FUNCTION_BLOCK AX_RF_TRIG (* Boolean falling and rising edge detection *)
  (* Standard: 61499-1 Annex A; Description: Copyright (c) 2017 fortiss GmbH, HR Agrartechnik GmbH This program and the accompanying materials are made available under the terms of the Eclipse Public License 2.0 which is available at https://www.eclipse.org/legal/epl-2.0/ SPDX-License-Identifier: EPL-2.0 *)
  (* Version 1.0, 2026-05-08, Franz Höpfinger, HR Agrartechnik GmbH, initial API and implementation and/or initial documentation *)
  PACKAGE adapter::events::unidirectional;
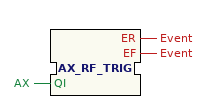
  EVENT_OUTPUT
    ER; (* confirmation that a rising edge was detected *)
    EF; (* confirmation that a falling edge was detected *)
  END_EVENT
  SOCKETS
    QI : adapter::types::unidirectional::AX; (* value to check for a rising or falling edge *)
  END_SOCKETS
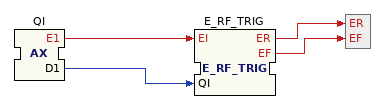
  FBS
    E_RF_TRIG : iec61499::events::E_RF_TRIG;
  END_FBS
  EVENT_CONNECTIONS
    QI.E1 TO E_RF_TRIG.EI;
    E_RF_TRIG.ER TO ER;
    E_RF_TRIG.EF TO EF;
  END_CONNECTIONS
  DATA_CONNECTIONS
    QI.D1 TO E_RF_TRIG.QI;
  END_CONNECTIONS
END_FUNCTION_BLOCK
